FUNCTION_BLOCK ASRT_3EVENTS_TO_SRT (* Composite FB for convert 3 EVENTS to ASRT *)
  (* Standard: 61499-2; Description: Copyright (c) 2026 HR Agrartechnik GmbH This program and the accompanying materials are made available under the terms of the Eclipse Public License 2.0 which is available at https://www.eclipse.org/legal/epl-2.0/ SPDX-License-Identifier: EPL-2.0 *)
  (* Version 1.0, 2026-09-03, Franz Höpfinger, HR Agrartechnik GmbH *)
  PACKAGE adapter::conversion::unidirectional;
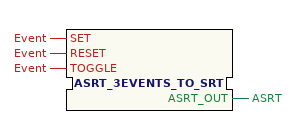
  EVENT_INPUT
    SET; (* Set / Switch on *)
    RESET; (* Reset / Switch off *)
    TOGGLE; (* Toggle / Switch output *)
  END_EVENT
  PLUGS
    ASRT_OUT : adapter::types::unidirectional::ASRT; (* Adapter Output *)
  END_PLUGS
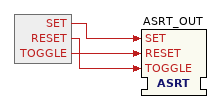
  EVENT_CONNECTIONS
    SET TO ASRT_OUT.SET;
    RESET TO ASRT_OUT.RESET;
    TOGGLE TO ASRT_OUT.TOGGLE;
  END_CONNECTIONS
END_FUNCTION_BLOCK
